FUNCTION HPF_FilterInit : REAL
VAR_INPUT
	CutFreq : REAL;
	Filter : POINTER TO HighPassFilter;
	TS : REAL;
END_VAR
VAR
END_VAR

	Filter^.FrequencyCut := CutFreq;
	Filter^.CutFreq := 1/1/(2*3.1415*Filter^.FrequencyCut);
	
	Filter^.Den := 1/(TS + 2*(Filter^.CutFreq));	
	
	
	Filter^.a1 := (TS-2*Filter^.CutFreq)*Filter^.Den;
	Filter^.b0 := (2*Filter^.CutFreq)*Filter^.Den;
	Filter^.b1 := -(2*Filter^.CutFreq)*Filter^.Den;

END_FUNCTION

(* stored: Version 1.1.0.1, ProductVersion 3.1.4024.4
   POU HPF_FilterInit: Id {9d310c2f-1456-4ec7-acee-f0b5066f55d0}, SpecialFunc None *)
